FUNCTION_BLOCK FB_MruInterface
VAR_INPUT
END_VAR
VAR_OUTPUT
END_VAR
VAR
	// Udp related
	{attribute 'tc_no_symbol'}
	udpServer : FB_UdpServer(0, 0, 0, 0, 0); // Dummy constructor
	{attribute 'tc_no_symbol'}
	rxUdp : ST_RxMru;



	
END_VAR

// Update udpServer
udpServer();

// Swap bytes of float data
BigToLittleEndian(ADR(rxUdp), SIZEOF(rxUdp));

METHOD BigToLittleEndian : BOOL
VAR_INPUT
	pData : PVOID;
	nData : UINT;
END_VAR



VAR
	pLE : PVOID;
	n : UINT;
	pOffset : UINT;
	bytesBE : ARRAY [0..3] OF BYTE;
	bytesLE : ARRAY [0..3] OF BYTE;
END_VAR
// NOTE: Only works with ST_RxMru struct!!! Not a genral function

FOR n := 0 TO (nData/4 - 2) DO
	// Current pointer offset index
	pOffset := 3 + 4*n;
	
	// Swap bytes
	IF pOffset <= nData THEN
		MEMCPY(ADR(bytesBE), pData + pOffset, 4);
	
		bytesLE[3] := bytesBE[0];
		bytesLE[2] := bytesBE[1];
		bytesLE[1] := bytesBE[2];
		bytesLE[0] := bytesBE[3];
		
		MEMCPY(pData + pOffset, ADR(bytesLE), 4);
	END_IF
END_FOR
END_METHOD

METHOD FB_exit : BOOL
VAR_INPUT
	bInCopyCode : BOOL; // if TRUE, the exit method is called for exiting an instance that is copied afterwards (online change).
END_VAR
END_METHOD

METHOD FB_init : BOOL
VAR_INPUT
	bInitRetains : BOOL; // if TRUE, the retain variables are initialized (warm start / cold start)
	bInCopyCode : BOOL;  // if TRUE, the instance afterwards gets moved into the copy code (online change)
	
	// Init variables
	_localPort : UINT;
END_VAR
// Initilize the udpServer
udpServer.FB_init(
	bInitRetains,
	bInCopyCode,
	_localPort,
	SIZEOF(rxUdp),
	ADR(rxUdp),
	0,
	0
);
END_METHOD

METHOD FB_reinit : BOOL
VAR_INPUT
END_VAR
END_METHOD

END_FUNCTION_BLOCK

(* stored: Version 1.1.0.1, ProductVersion 3.1.4022.7
   POU FB_MruInterface: Id {c6b5539c-66b4-48be-8e8d-e330098c72f8}, SpecialFunc None
   Method BigToLittleEndian: Id {55be5d21-786e-44c3-a382-2ff80affc77c}
   Method FB_exit: Id {a3e9d2a2-7999-4f51-bfdc-9869126d272a}
   Method FB_init: Id {3130c499-1695-4075-b5a0-733165c80fd1}
   Method FB_reinit: Id {1faf6911-8283-46ae-9bd2-81f20ae258ae} *)
